// ---- AnalogIO/Outputs/EL4022/EL4022_EX.TcDUT
(*
SPDX-FileCopyrightText: © 2026 Oleksandr Tiutyk <trofimich@gmail.com>
SPDX-License-Identifier: MIT
License: https://opensource.org/license/mit
*)

(*!
<summary>
Beckhoff EL4022_EX: Extended 2-channel analog output terminal (4 .. 20 mA, 12-bit) with diagnostics.
</summary>
<description>
Extends EL4022 with EtherCAT Working Counter, slave state, and CoE mailbox ADS address diagnostics.
When used for I/O, link located fields or their containing buffers to the matching selected PDOs.
The record is not a packed wire buffer; compiler padding is not part of the device specification.
Unlinked/default values do not prove valid I/O. The caller evaluates bus/channel validity before use.
Use one owner task per instance and externally synchronize other access; multi-field snapshots are not atomic.
Copies store data without creating hardware links. Keep borrowed field references valid while consumers are bound.
This passive record performs no validation, synchronization, configuration or protocol advancement.
WcState=TRUE means process-data exchange is invalid. State is acyclic EtherCAT/link information,
not proof of current measurement validity. Link diagnostics to the matching slave InfoData entries.
The selected PDO representation is documented by the base terminal model.
AdsAddr is acyclic mailbox addressing information, not a measurement-validity indicator.
Channels hold raw INT16 output commands; configure electrical range and presentation before use.
</description>
*)
TYPE EL4022_EX EXTENDS EL4022 :
STRUCT
	WcState AT %I* : BOOL;
	State AT %I* : UINT;
	AdsAddr AT %I* : Global.AMSADDR;
END_STRUCT
END_TYPE

// ---- AnalogIO/Outputs/EL4024/EL4024.TcDUT
(*
SPDX-FileCopyrightText: © 2026 Oleksandr Tiutyk <trofimich@gmail.com>
SPDX-License-Identifier: MIT
License: https://opensource.org/license/mit
*)

(*!
<summary>
Beckhoff EL4024: 4-channel analog output terminal (4 .. 20 mA, 12-bit).
</summary>
<description>
Process image mapping structure for the EL4024 EtherCAT terminal with 4 analog output channel(s).
When used for I/O, link located fields or their containing buffers to the matching selected PDOs.
The record is not a packed wire buffer; compiler padding is not part of the device specification.
Unlinked/default values do not prove valid I/O. The caller evaluates bus/channel validity before use.
Use one owner task per instance and externally synchronize other access; multi-field snapshots are not atomic.
Copies store data without creating hardware links. Keep borrowed field references valid while consumers are bound.
This passive record performs no validation, synchronization, configuration or protocol advancement.
Channels hold raw INT16 output commands; configure electrical range and presentation before use.
</description>
*)
TYPE EL4024 :
STRUCT
	Ch1 AT %Q* : INT;
	Ch2 AT %Q* : INT;
	Ch3 AT %Q* : INT;
	Ch4 AT %Q* : INT;
END_STRUCT
END_TYPE

// ---- AnalogIO/Outputs/EL4024/EL4024_EX.TcDUT
(*
SPDX-FileCopyrightText: © 2026 Oleksandr Tiutyk <trofimich@gmail.com>
SPDX-License-Identifier: MIT
License: https://opensource.org/license/mit
*)

(*!
<summary>
Beckhoff EL4024_EX: Extended 4-channel analog output terminal (4 .. 20 mA, 12-bit) with diagnostics.
</summary>
<description>
Extends EL4024 with EtherCAT Working Counter, slave state, and CoE mailbox ADS address diagnostics.
When used for I/O, link located fields or their containing buffers to the matching selected PDOs.
The record is not a packed wire buffer; compiler padding is not part of the device specification.
Unlinked/default values do not prove valid I/O. The caller evaluates bus/channel validity before use.
Use one owner task per instance and externally synchronize other access; multi-field snapshots are not atomic.
Copies store data without creating hardware links. Keep borrowed field references valid while consumers are bound.
This passive record performs no validation, synchronization, configuration or protocol advancement.
WcState=TRUE means process-data exchange is invalid. State is acyclic EtherCAT/link information,
not proof of current measurement validity. Link diagnostics to the matching slave InfoData entries.
The selected PDO representation is documented by the base terminal model.
AdsAddr is acyclic mailbox addressing information, not a measurement-validity indicator.
Channels hold raw INT16 output commands; configure electrical range and presentation before use.
</description>
*)
TYPE EL4024_EX EXTENDS EL4024 :
STRUCT
	WcState AT %I* : BOOL;
	State AT %I* : UINT;
	AdsAddr AT %I* : Global.AMSADDR;
END_STRUCT
END_TYPE

// ---- AnalogIO/Outputs/EL4028/EL4028.TcDUT
(*
SPDX-FileCopyrightText: © 2026 Oleksandr Tiutyk <trofimich@gmail.com>
SPDX-License-Identifier: MIT
License: https://opensource.org/license/mit
*)

(*!
<summary>
Beckhoff EL4028: 8-channel analog output terminal (4 .. 20 mA, 12-bit).
</summary>
<description>
Process image mapping structure for the EL4028 EtherCAT terminal with 8 analog output channel(s).
When used for I/O, link located fields or their containing buffers to the matching selected PDOs.
The record is not a packed wire buffer; compiler padding is not part of the device specification.
Unlinked/default values do not prove valid I/O. The caller evaluates bus/channel validity before use.
Use one owner task per instance and externally synchronize other access; multi-field snapshots are not atomic.
Copies store data without creating hardware links. Keep borrowed field references valid while consumers are bound.
This passive record performs no validation, synchronization, configuration or protocol advancement.
Channels hold raw INT16 output commands; configure electrical range and presentation before use.
</description>
*)
TYPE EL4028 :
STRUCT
	Ch1 AT %Q* : INT;
	Ch2 AT %Q* : INT;
	Ch3 AT %Q* : INT;
	Ch4 AT %Q* : INT;
	Ch5 AT %Q* : INT;
	Ch6 AT %Q* : INT;
	Ch7 AT %Q* : INT;
	Ch8 AT %Q* : INT;
END_STRUCT
END_TYPE

// ---- AnalogIO/Outputs/EL4028/EL4028_EX.TcDUT
(*
SPDX-FileCopyrightText: © 2026 Oleksandr Tiutyk <trofimich@gmail.com>
SPDX-License-Identifier: MIT
License: https://opensource.org/license/mit
*)

(*!
<summary>
Beckhoff EL4028_EX: Extended 8-channel analog output terminal (4 .. 20 mA, 12-bit) with diagnostics.
</summary>
<description>
Extends EL4028 with EtherCAT Working Counter, slave state, and CoE mailbox ADS address diagnostics.
When used for I/O, link located fields or their containing buffers to the matching selected PDOs.
The record is not a packed wire buffer; compiler padding is not part of the device specification.
Unlinked/default values do not prove valid I/O. The caller evaluates bus/channel validity before use.
Use one owner task per instance and externally synchronize other access; multi-field snapshots are not atomic.
Copies store data without creating hardware links. Keep borrowed field references valid while consumers are bound.
This passive record performs no validation, synchronization, configuration or protocol advancement.
WcState=TRUE means process-data exchange is invalid. State is acyclic EtherCAT/link information,
not proof of current measurement validity. Link diagnostics to the matching slave InfoData entries.
The selected PDO representation is documented by the base terminal model.
AdsAddr is acyclic mailbox addressing information, not a measurement-validity indicator.
Channels hold raw INT16 output commands; configure electrical range and presentation before use.
</description>
*)
TYPE EL4028_EX EXTENDS EL4028 :
STRUCT
	WcState AT %I* : BOOL;
	State AT %I* : UINT;
	AdsAddr AT %I* : Global.AMSADDR;
END_STRUCT
END_TYPE

// ---- AnalogIO/Outputs/EL4102/EL4102.TcDUT
(*
SPDX-FileCopyrightText: © 2026 Oleksandr Tiutyk <trofimich@gmail.com>
SPDX-License-Identifier: MIT
License: https://opensource.org/license/mit
*)

(*!
<summary>
Beckhoff EL4102: 2-channel analog output terminal (0 .. 10 V, 16-bit).
</summary>
<description>
Process image mapping structure for the EL4102 EtherCAT terminal with 2 analog output channel(s).
When used for I/O, link located fields or their containing buffers to the matching selected PDOs.
The record is not a packed wire buffer; compiler padding is not part of the device specification.
Unlinked/default values do not prove valid I/O. The caller evaluates bus/channel validity before use.
Use one owner task per instance and externally synchronize other access; multi-field snapshots are not atomic.
Copies store data without creating hardware links. Keep borrowed field references valid while consumers are bound.
This passive record performs no validation, synchronization, configuration or protocol advancement.
Channels hold raw INT16 output commands; configure electrical range and presentation before use.
</description>
*)
TYPE EL4102 :
STRUCT
	Ch1 AT %Q* : INT;
	Ch2 AT %Q* : INT;
END_STRUCT
END_TYPE

// ---- AnalogIO/Outputs/EL4102/EL4102_EX.TcDUT
(*
SPDX-FileCopyrightText: © 2026 Oleksandr Tiutyk <trofimich@gmail.com>
SPDX-License-Identifier: MIT
License: https://opensource.org/license/mit
*)

(*!
<summary>
Beckhoff EL4102_EX: Extended 2-channel analog output terminal (0 .. 10 V, 16-bit) with diagnostics.
</summary>
<description>
Extends EL4102 with EtherCAT Working Counter, slave state, and CoE mailbox ADS address diagnostics.
When used for I/O, link located fields or their containing buffers to the matching selected PDOs.
The record is not a packed wire buffer; compiler padding is not part of the device specification.
Unlinked/default values do not prove valid I/O. The caller evaluates bus/channel validity before use.
Use one owner task per instance and externally synchronize other access; multi-field snapshots are not atomic.
Copies store data without creating hardware links. Keep borrowed field references valid while consumers are bound.
This passive record performs no validation, synchronization, configuration or protocol advancement.
WcState=TRUE means process-data exchange is invalid. State is acyclic EtherCAT/link information,
not proof of current measurement validity. Link diagnostics to the matching slave InfoData entries.
The selected PDO representation is documented by the base terminal model.
AdsAddr is acyclic mailbox addressing information, not a measurement-validity indicator.
Channels hold raw INT16 output commands; configure electrical range and presentation before use.
</description>
*)
TYPE EL4102_EX EXTENDS EL4102 :
STRUCT
	WcState AT %I* : BOOL;
	State AT %I* : UINT;
	AdsAddr AT %I* : Global.AMSADDR;
END_STRUCT
END_TYPE

// ---- AnalogIO/Outputs/EL4104/EL4104.TcDUT
(*
SPDX-FileCopyrightText: © 2026 Oleksandr Tiutyk <trofimich@gmail.com>
SPDX-License-Identifier: MIT
License: https://opensource.org/license/mit
*)

(*!
<summary>
Beckhoff EL4104: 4-channel analog output terminal (0 .. 10 V, 16-bit).
</summary>
<description>
Process image mapping structure for the EL4104 EtherCAT terminal with 4 analog output channel(s).
When used for I/O, link located fields or their containing buffers to the matching selected PDOs.
The record is not a packed wire buffer; compiler padding is not part of the device specification.
Unlinked/default values do not prove valid I/O. The caller evaluates bus/channel validity before use.
Use one owner task per instance and externally synchronize other access; multi-field snapshots are not atomic.
Copies store data without creating hardware links. Keep borrowed field references valid while consumers are bound.
This passive record performs no validation, synchronization, configuration or protocol advancement.
Channels hold raw INT16 output commands; configure electrical range and presentation before use.
</description>
*)
TYPE EL4104 :
STRUCT
	Ch1 AT %Q* : INT;
	Ch2 AT %Q* : INT;
	Ch3 AT %Q* : INT;
	Ch4 AT %Q* : INT;
END_STRUCT
END_TYPE

// ---- AnalogIO/Outputs/EL4104/EL4104_EX.TcDUT
(*
SPDX-FileCopyrightText: © 2026 Oleksandr Tiutyk <trofimich@gmail.com>
SPDX-License-Identifier: MIT
License: https://opensource.org/license/mit
*)

(*!
<summary>
Beckhoff EL4104_EX: Extended 4-channel analog output terminal (0 .. 10 V, 16-bit) with diagnostics.
</summary>
<description>
Extends EL4104 with EtherCAT Working Counter, slave state, and CoE mailbox ADS address diagnostics.
When used for I/O, link located fields or their containing buffers to the matching selected PDOs.
The record is not a packed wire buffer; compiler padding is not part of the device specification.
Unlinked/default values do not prove valid I/O. The caller evaluates bus/channel validity before use.
Use one owner task per instance and externally synchronize other access; multi-field snapshots are not atomic.
Copies store data without creating hardware links. Keep borrowed field references valid while consumers are bound.
This passive record performs no validation, synchronization, configuration or protocol advancement.
WcState=TRUE means process-data exchange is invalid. State is acyclic EtherCAT/link information,
not proof of current measurement validity. Link diagnostics to the matching slave InfoData entries.
The selected PDO representation is documented by the base terminal model.
AdsAddr is acyclic mailbox addressing information, not a measurement-validity indicator.
Channels hold raw INT16 output commands; configure electrical range and presentation before use.
</description>
*)
TYPE EL4104_EX EXTENDS EL4104 :
STRUCT
	WcState AT %I* : BOOL;
	State AT %I* : UINT;
	AdsAddr AT %I* : Global.AMSADDR;
END_STRUCT
END_TYPE

// ---- AnalogIO/Outputs/EL4132/EL4132.TcDUT
(*
SPDX-FileCopyrightText: © 2026 Oleksandr Tiutyk <trofimich@gmail.com>
SPDX-License-Identifier: MIT
License: https://opensource.org/license/mit
*)

(*!
<summary>
Beckhoff EL4132: 2-channel analog output terminal (-10 V .. +10 V, 16-bit).
</summary>
<description>
Process image mapping structure for the EL4132 EtherCAT terminal with 2 analog output channel(s).
When used for I/O, link located fields or their containing buffers to the matching selected PDOs.
The record is not a packed wire buffer; compiler padding is not part of the device specification.
Unlinked/default values do not prove valid I/O. The caller evaluates bus/channel validity before use.
Use one owner task per instance and externally synchronize other access; multi-field snapshots are not atomic.
Copies store data without creating hardware links. Keep borrowed field references valid while consumers are bound.
This passive record performs no validation, synchronization, configuration or protocol advancement.
Channels hold raw INT16 output commands; configure electrical range and presentation before use.
</description>
*)
TYPE EL4132 :
STRUCT
	Ch1 AT %Q* : INT;
	Ch2 AT %Q* : INT;
END_STRUCT
END_TYPE

// ---- AnalogIO/Outputs/EL4132/EL4132_EX.TcDUT
(*
SPDX-FileCopyrightText: © 2026 Oleksandr Tiutyk <trofimich@gmail.com>
SPDX-License-Identifier: MIT
License: https://opensource.org/license/mit
*)

(*!
<summary>
Beckhoff EL4132_EX: Extended 2-channel analog output terminal (-10 V .. +10 V, 16-bit) with diagnostics.
</summary>
<description>
Extends EL4132 with EtherCAT Working Counter, slave state, and CoE mailbox ADS address diagnostics.
When used for I/O, link located fields or their containing buffers to the matching selected PDOs.
The record is not a packed wire buffer; compiler padding is not part of the device specification.
Unlinked/default values do not prove valid I/O. The caller evaluates bus/channel validity before use.
Use one owner task per instance and externally synchronize other access; multi-field snapshots are not atomic.
Copies store data without creating hardware links. Keep borrowed field references valid while consumers are bound.
This passive record performs no validation, synchronization, configuration or protocol advancement.
WcState=TRUE means process-data exchange is invalid. State is acyclic EtherCAT/link information,
not proof of current measurement validity. Link diagnostics to the matching slave InfoData entries.
The selected PDO representation is documented by the base terminal model.
AdsAddr is acyclic mailbox addressing information, not a measurement-validity indicator.
Channels hold raw INT16 output commands; configure electrical range and presentation before use.
</description>
*)
TYPE EL4132_EX EXTENDS EL4132 :
STRUCT
	WcState AT %I* : BOOL;
	State AT %I* : UINT;
	AdsAddr AT %I* : Global.AMSADDR;
END_STRUCT
END_TYPE

// ---- AnalogIO/Outputs/EL4134/EL4134.TcDUT
(*
SPDX-FileCopyrightText: © 2026 Oleksandr Tiutyk <trofimich@gmail.com>
SPDX-License-Identifier: MIT
License: https://opensource.org/license/mit
*)

(*!
<summary>
Beckhoff EL4134: 4-channel analog output terminal (-10 V .. +10 V, 16-bit).
</summary>
<description>
Process image mapping structure for the EL4134 EtherCAT terminal with 4 analog output channel(s).
When used for I/O, link located fields or their containing buffers to the matching selected PDOs.
The record is not a packed wire buffer; compiler padding is not part of the device specification.
Unlinked/default values do not prove valid I/O. The caller evaluates bus/channel validity before use.
Use one owner task per instance and externally synchronize other access; multi-field snapshots are not atomic.
Copies store data without creating hardware links. Keep borrowed field references valid while consumers are bound.
This passive record performs no validation, synchronization, configuration or protocol advancement.
Channels hold raw INT16 output commands; configure electrical range and presentation before use.
</description>
*)
TYPE EL4134 :
STRUCT
	Ch1 AT %Q* : INT;
	Ch2 AT %Q* : INT;
	Ch3 AT %Q* : INT;
	Ch4 AT %Q* : INT;
END_STRUCT
END_TYPE

// ---- AnalogIO/Outputs/EL4134/EL4134_EX.TcDUT
(*
SPDX-FileCopyrightText: © 2026 Oleksandr Tiutyk <trofimich@gmail.com>
SPDX-License-Identifier: MIT
License: https://opensource.org/license/mit
*)

(*!
<summary>
Beckhoff EL4134_EX: Extended 4-channel analog output terminal (-10 V .. +10 V, 16-bit) with diagnostics.
</summary>
<description>
Extends EL4134 with EtherCAT Working Counter, slave state, and CoE mailbox ADS address diagnostics.
When used for I/O, link located fields or their containing buffers to the matching selected PDOs.
The record is not a packed wire buffer; compiler padding is not part of the device specification.
Unlinked/default values do not prove valid I/O. The caller evaluates bus/channel validity before use.
Use one owner task per instance and externally synchronize other access; multi-field snapshots are not atomic.
Copies store data without creating hardware links. Keep borrowed field references valid while consumers are bound.
This passive record performs no validation, synchronization, configuration or protocol advancement.
WcState=TRUE means process-data exchange is invalid. State is acyclic EtherCAT/link information,
not proof of current measurement validity. Link diagnostics to the matching slave InfoData entries.
The selected PDO representation is documented by the base terminal model.
AdsAddr is acyclic mailbox addressing information, not a measurement-validity indicator.
Channels hold raw INT16 output commands; configure electrical range and presentation before use.
</description>
*)
TYPE EL4134_EX EXTENDS EL4134 :
STRUCT
	WcState AT %I* : BOOL;
	State AT %I* : UINT;
	AdsAddr AT %I* : Global.AMSADDR;
END_STRUCT
END_TYPE

// ---- AnalogIO/Outputs/EL4122/EL4122.TcDUT
(*
SPDX-FileCopyrightText: © 2026 Oleksandr Tiutyk <trofimich@gmail.com>
SPDX-License-Identifier: MIT
License: https://opensource.org/license/mit
*)

(*!
<summary>
Beckhoff EL4122: 2-channel analog output terminal (4 .. 20 mA, 16-bit).
</summary>
<description>
Process image mapping structure for the EL4122 EtherCAT terminal with 2 analog output channel(s).
When used for I/O, link located fields or their containing buffers to the matching selected PDOs.
The record is not a packed wire buffer; compiler padding is not part of the device specification.
Unlinked/default values do not prove valid I/O. The caller evaluates bus/channel validity before use.
Use one owner task per instance and externally synchronize other access; multi-field snapshots are not atomic.
Copies store data without creating hardware links. Keep borrowed field references valid while consumers are bound.
This passive record performs no validation, synchronization, configuration or protocol advancement.
Channels hold raw INT16 output commands; configure electrical range and presentation before use.
</description>
*)
TYPE EL4122 :
STRUCT
	Ch1 AT %Q* : INT;
	Ch2 AT %Q* : INT;
END_STRUCT
END_TYPE

// ---- AnalogIO/Outputs/EL4122/EL4122_EX.TcDUT
(*
SPDX-FileCopyrightText: © 2026 Oleksandr Tiutyk <trofimich@gmail.com>
SPDX-License-Identifier: MIT
License: https://opensource.org/license/mit
*)

(*!
<summary>
Beckhoff EL4122_EX: Extended 2-channel analog output terminal (4 .. 20 mA, 16-bit) with diagnostics.
</summary>
<description>
Extends EL4122 with EtherCAT Working Counter, slave state, and CoE mailbox ADS address diagnostics.
When used for I/O, link located fields or their containing buffers to the matching selected PDOs.
The record is not a packed wire buffer; compiler padding is not part of the device specification.
Unlinked/default values do not prove valid I/O. The caller evaluates bus/channel validity before use.
Use one owner task per instance and externally synchronize other access; multi-field snapshots are not atomic.
Copies store data without creating hardware links. Keep borrowed field references valid while consumers are bound.
This passive record performs no validation, synchronization, configuration or protocol advancement.
WcState=TRUE means process-data exchange is invalid. State is acyclic EtherCAT/link information,
not proof of current measurement validity. Link diagnostics to the matching slave InfoData entries.
The selected PDO representation is documented by the base terminal model.
AdsAddr is acyclic mailbox addressing information, not a measurement-validity indicator.
Channels hold raw INT16 output commands; configure electrical range and presentation before use.
</description>
*)
TYPE EL4122_EX EXTENDS EL4122 :
STRUCT
	WcState AT %I* : BOOL;
	State AT %I* : UINT;
	AdsAddr AT %I* : Global.AMSADDR;
END_STRUCT
END_TYPE

// ---- AnalogIO/Outputs/EL4124/EL4124.TcDUT
(*
SPDX-FileCopyrightText: © 2026 Oleksandr Tiutyk <trofimich@gmail.com>
SPDX-License-Identifier: MIT
License: https://opensource.org/license/mit
*)

(*!
<summary>
Beckhoff EL4124: 4-channel analog output terminal (4 .. 20 mA, 16-bit).
</summary>
<description>
Process image mapping structure for the EL4124 EtherCAT terminal with 4 analog output channel(s).
When used for I/O, link located fields or their containing buffers to the matching selected PDOs.
The record is not a packed wire buffer; compiler padding is not part of the device specification.
Unlinked/default values do not prove valid I/O. The caller evaluates bus/channel validity before use.
Use one owner task per instance and externally synchronize other access; multi-field snapshots are not atomic.
Copies store data without creating hardware links. Keep borrowed field references valid while consumers are bound.
This passive record performs no validation, synchronization, configuration or protocol advancement.
Channels hold raw INT16 output commands; configure electrical range and presentation before use.
</description>
*)
TYPE EL4124 :
STRUCT
	Ch1 AT %Q* : INT;
	Ch2 AT %Q* : INT;
	Ch3 AT %Q* : INT;
	Ch4 AT %Q* : INT;
END_STRUCT
END_TYPE

// ---- AnalogIO/Outputs/EL4124/EL4124_EX.TcDUT
(*
SPDX-FileCopyrightText: © 2026 Oleksandr Tiutyk <trofimich@gmail.com>
SPDX-License-Identifier: MIT
License: https://opensource.org/license/mit
*)

(*!
<summary>
Beckhoff EL4124_EX: Extended 4-channel analog output terminal (4 .. 20 mA, 16-bit) with diagnostics.
</summary>
<description>
Extends EL4124 with EtherCAT Working Counter, slave state, and CoE mailbox ADS address diagnostics.
When used for I/O, link located fields or their containing buffers to the matching selected PDOs.
The record is not a packed wire buffer; compiler padding is not part of the device specification.
Unlinked/default values do not prove valid I/O. The caller evaluates bus/channel validity before use.
Use one owner task per instance and externally synchronize other access; multi-field snapshots are not atomic.
Copies store data without creating hardware links. Keep borrowed field references valid while consumers are bound.
This passive record performs no validation, synchronization, configuration or protocol advancement.
WcState=TRUE means process-data exchange is invalid. State is acyclic EtherCAT/link information,
not proof of current measurement validity. Link diagnostics to the matching slave InfoData entries.
The selected PDO representation is documented by the base terminal model.
AdsAddr is acyclic mailbox addressing information, not a measurement-validity indicator.
Channels hold raw INT16 output commands; configure electrical range and presentation before use.
</description>
*)
TYPE EL4124_EX EXTENDS EL4124 :
STRUCT
	WcState AT %I* : BOOL;
	State AT %I* : UINT;
	AdsAddr AT %I* : Global.AMSADDR;
END_STRUCT
END_TYPE

// ---- Weighing/STRAIN_GAUGE_INPUT_CHANNEL.TcDUT
(*
SPDX-FileCopyrightText: © 2026 Oleksandr Tiutyk <trofimich@gmail.com>
SPDX-License-Identifier: MIT
License: https://opensource.org/license/mit
*)

(*!
<summary>
Beckhoff strain gauge / resistor bridge input channel process image.
</summary>
<description>
Represents EL3356/EL3356-0010 input PDO 0x1A00 with 16-bit Status and PDO 0x1A01 with signed 32-bit Value.
Both input PDOs are required. Link Status to RMB Status and Value to RMB Value (INT32) separately;
PDO 0x1A01 alone does not contain status information.
Select the integer assignment; REAL load and two-channel voltage modes require different types.
Calibration and device settings determine engineering scaling. Evaluate Status before using Value.
When used for I/O, link located fields or their containing buffers to the matching selected PDOs.
The record is not a packed wire buffer; compiler padding is not part of the device specification.
Unlinked/default values do not prove valid I/O. The caller evaluates bus/channel validity before use.
Use one owner task per instance and externally synchronize other access; multi-field snapshots are not atomic.
Copies store data without creating hardware links. Keep borrowed field references valid while consumers are bound.
This passive record performs no validation, synchronization, configuration or protocol advancement.
</description>
*)
TYPE STRAIN_GAUGE_INPUT_CHANNEL :
STRUCT
	Status AT %I* : WORD;
	Value AT %I* : DINT;
END_STRUCT
END_TYPE

// ---- Weighing/STRAIN_GAUGE_OUTPUT_CHANNEL.TcDUT
(*
SPDX-FileCopyrightText: © 2026 Oleksandr Tiutyk <trofimich@gmail.com>
SPDX-License-Identifier: MIT
License: https://opensource.org/license/mit
*)

(*!
<summary>
Beckhoff strain gauge / resistor bridge output control channel process image.
</summary>
<description>
Encapsulates a 16-bit control word for calibration, tare, and filtering commands on measuring bridge terminals
(e.g. EL3356).
When used for I/O, link located fields or their containing buffers to the matching selected PDOs.
The record is not a packed wire buffer; compiler padding is not part of the device specification.
Unlinked/default values do not prove valid I/O. The caller evaluates bus/channel validity before use.
Use one owner task per instance and externally synchronize other access; multi-field snapshots are not atomic.
Copies store data without creating hardware links. Keep borrowed field references valid while consumers are bound.
This passive record performs no validation, synchronization, configuration or protocol advancement.
</description>
*)
TYPE STRAIN_GAUGE_OUTPUT_CHANNEL :
STRUCT
	Control AT %Q* : WORD;
END_STRUCT
END_TYPE

// ---- Weighing/STRAIN_GAUGE_CHANNEL.TcDUT
(*
SPDX-FileCopyrightText: © 2026 Oleksandr Tiutyk <trofimich@gmail.com>
SPDX-License-Identifier: MIT
License: https://opensource.org/license/mit
*)

(*!
<summary>
Beckhoff bidirectional strain gauge / resistor bridge channel process image.
</summary>
<description>
Aggregates input status/value (STRAIN_GAUGE_INPUT_CHANNEL) and output control (STRAIN_GAUGE_OUTPUT_CHANNEL)
for one measuring bridge channel.
When used for I/O, link located fields or their containing buffers to the matching selected PDOs.
The record is not a packed wire buffer; compiler padding is not part of the device specification.
Unlinked/default values do not prove valid I/O. The caller evaluates bus/channel validity before use.
Use one owner task per instance and externally synchronize other access; multi-field snapshots are not atomic.
Copies store data without creating hardware links. Keep borrowed field references valid while consumers are bound.
This passive record performs no validation, synchronization, configuration or protocol advancement.
</description>
*)
TYPE STRAIN_GAUGE_CHANNEL :
STRUCT
	In : STRAIN_GAUGE_INPUT_CHANNEL;
	Out : STRAIN_GAUGE_OUTPUT_CHANNEL;
END_STRUCT
END_TYPE

// ---- Weighing/EL3356/EL3356.TcDUT
(*
SPDX-FileCopyrightText: © 2026 Oleksandr Tiutyk <trofimich@gmail.com>
SPDX-License-Identifier: MIT
License: https://opensource.org/license/mit
*)

(*!
<summary>
Beckhoff EL3356: 1-channel precise resistor bridge / load cell terminal (24-bit).
</summary>
<description>
Requires the one-channel strain-gauge INT32 assignment: status PDO 0x1A00, value PDO 0x1A01,
and control PDO 0x1600. Keep both input PDOs enabled and link Status and Value separately.
Value is signed calculated load; engineering scaling follows calibration. REAL load, two-channel voltage,
optional filter-frequency and timestamp PDOs are outside this model; disable or link optional PDOs separately.
When used for I/O, link located fields or their containing buffers to the matching selected PDOs.
The record is not a packed wire buffer; compiler padding is not part of the device specification.
Unlinked/default values do not prove valid I/O. The caller evaluates bus/channel validity before use.
Use one owner task per instance and externally synchronize other access; multi-field snapshots are not atomic.
Copies store data without creating hardware links. Keep borrowed field references valid while consumers are bound.
This passive record performs no validation, synchronization, configuration or protocol advancement.
</description>
*)
TYPE EL3356 :
STRUCT
	Ch1 : STRAIN_GAUGE_CHANNEL;
END_STRUCT
END_TYPE

// ---- Weighing/EL3356/EL3356_EX.TcDUT
(*
SPDX-FileCopyrightText: © 2026 Oleksandr Tiutyk <trofimich@gmail.com>
SPDX-License-Identifier: MIT
License: https://opensource.org/license/mit
*)

(*!
<summary>
Beckhoff EL3356_EX: Extended 1-channel load cell terminal with diagnostics.
</summary>
<description>
Extends EL3356 with EtherCAT Working Counter, slave state, and CoE mailbox ADS address diagnostics.
When used for I/O, link located fields or their containing buffers to the matching selected PDOs.
The record is not a packed wire buffer; compiler padding is not part of the device specification.
Unlinked/default values do not prove valid I/O. The caller evaluates bus/channel validity before use.
Use one owner task per instance and externally synchronize other access; multi-field snapshots are not atomic.
Copies store data without creating hardware links. Keep borrowed field references valid while consumers are bound.
This passive record performs no validation, synchronization, configuration or protocol advancement.
WcState=TRUE means process-data exchange is invalid. State is acyclic EtherCAT/link information,
not proof of current measurement validity. Link diagnostics to the matching slave InfoData entries.
The selected PDO representation is documented by the base terminal model.
InputToggle signals an input update by changing state; TRUE alone does not mean fresh data.
AdsAddr is acyclic mailbox addressing information, not a measurement-validity indicator.
</description>
*)
TYPE EL3356_EX EXTENDS EL3356 :
STRUCT
	WcState AT %I* : BOOL;
	InputToggle AT %I* : BOOL;
	State AT %I* : UINT;
	AdsAddr AT %I* : Global.AMSADDR;
END_STRUCT
END_TYPE

// ---- Weighing/EL3356_0010/EL3356_0010.TcDUT
(*
SPDX-FileCopyrightText: © 2026 Oleksandr Tiutyk <trofimich@gmail.com>
SPDX-License-Identifier: MIT
License: https://opensource.org/license/mit
*)

(*!
<summary>
Beckhoff EL3356-0010: Fast 1-channel precise resistor bridge / load cell terminal with Distributed Clocks.
</summary>
<description>
Requires the one-channel strain-gauge INT32 assignment: status PDO 0x1A00, value PDO 0x1A01,
and control PDO 0x1600. Keep both input PDOs enabled and link Status and Value separately.
Value is signed calculated load; engineering scaling follows calibration. REAL load, two-channel voltage,
optional filter-frequency and timestamp PDOs are outside this model; disable or link optional PDOs separately.
When used for I/O, link located fields or their containing buffers to the matching selected PDOs.
The record is not a packed wire buffer; compiler padding is not part of the device specification.
Unlinked/default values do not prove valid I/O. The caller evaluates bus/channel validity before use.
Use one owner task per instance and externally synchronize other access; multi-field snapshots are not atomic.
Copies store data without creating hardware links. Keep borrowed field references valid while consumers are bound.
This passive record performs no validation, synchronization, configuration or protocol advancement.
</description>
*)
TYPE EL3356_0010 :
STRUCT
	Ch1 : STRAIN_GAUGE_CHANNEL;
END_STRUCT
END_TYPE

// ---- Weighing/EL3356_0010/EL3356_0010_EX.TcDUT
(*
SPDX-FileCopyrightText: © 2026 Oleksandr Tiutyk <trofimich@gmail.com>
SPDX-License-Identifier: MIT
License: https://opensource.org/license/mit
*)

(*!
<summary>
Beckhoff EL3356_0010_EX: Extended fast 1-channel load cell terminal with diagnostics.
</summary>
<description>
Extends EL3356_0010 with EtherCAT Working Counter, slave state, and CoE mailbox ADS address diagnostics.
When used for I/O, link located fields or their containing buffers to the matching selected PDOs.
The record is not a packed wire buffer; compiler padding is not part of the device specification.
Unlinked/default values do not prove valid I/O. The caller evaluates bus/channel validity before use.
Use one owner task per instance and externally synchronize other access; multi-field snapshots are not atomic.
Copies store data without creating hardware links. Keep borrowed field references valid while consumers are bound.
This passive record performs no validation, synchronization, configuration or protocol advancement.
WcState=TRUE means process-data exchange is invalid. State is acyclic EtherCAT/link information,
not proof of current measurement validity. Link diagnostics to the matching slave InfoData entries.
The selected PDO representation is documented by the base terminal model.
InputToggle signals an input update by changing state; TRUE alone does not mean fresh data.
AdsAddr is acyclic mailbox addressing information, not a measurement-validity indicator.
</description>
*)
TYPE EL3356_0010_EX EXTENDS EL3356_0010 :
STRUCT
	WcState AT %I* : BOOL;
	InputToggle AT %I* : BOOL;
	State AT %I* : UINT;
	AdsAddr AT %I* : Global.AMSADDR;
END_STRUCT
END_TYPE

// ---- PowerMeasurement/POWER_MEASUREMENT_INPUT_CHANNEL.TcDUT
(*
SPDX-FileCopyrightText: © 2026 Oleksandr Tiutyk <trofimich@gmail.com>
SPDX-License-Identifier: MIT
License: https://opensource.org/license/mit
*)

(*!
<summary>
Beckhoff 3-phase power measurement input channel process image.
</summary>
<description>
Represents EL3413/EL3433 phase PDO 0x1A00, 0x1A01 or 0x1A02, including mandatory channel Status.
Status contains voltage/current limits, phase sequence, missing zero crossing, TxPDO State and Toggle.
Reject data when Status bit 14 is set; bit 15 toggles on update. Evaluate bus validity as well.
Current is signed in 0.000001 A, Voltage in 0.0001 V and ActivePower in 0.01 W before transformer ratios.
Index acknowledges the selection for VariantValue; do not interpret it using only the requested output Index.
Indices 0..5 select apparent power (0.01 VA), reactive power (0.01 var), energy (0.001 Wh), power factor
(0.001), frequency (0.1 Hz) and negative energy (0.001 Wh). Further indices depend on device firmware.
EL3403 uses EL3403_INPUT_CHANNEL because its phase status differs. Link fields individually, not as a wire buffer.
Use one owner task and synchronize other access; copies do not guarantee an atomic snapshot.
When used for I/O, link located fields or their containing buffers to the matching selected PDOs.
The record is not a packed wire buffer; compiler padding is not part of the device specification.
Unlinked/default values do not prove valid I/O. The caller evaluates bus/channel validity before use.
Use one owner task per instance and externally synchronize other access; multi-field snapshots are not atomic.
Copies store data without creating hardware links. Keep borrowed field references valid while consumers are bound.
This passive record performs no validation, synchronization, configuration or protocol advancement.
</description>
*)
TYPE POWER_MEASUREMENT_INPUT_CHANNEL :
STRUCT
	//! <summary>Phase status; TxPDO State bit 14 invalidates data and bit 15 toggles on update.</summary>
	Status AT %I* : WORD;
	Current AT %I* : DINT;
	Voltage AT %I* : DINT;
	ActivePower AT %I* : DINT;
	Index AT %I* : USINT;
	VariantValue AT %I* : DINT;
END_STRUCT
END_TYPE

// ---- PowerMeasurement/POWER_MEASUREMENT_OUTPUT_CHANNEL.TcDUT
(*
SPDX-FileCopyrightText: © 2026 Oleksandr Tiutyk <trofimich@gmail.com>
SPDX-License-Identifier: MIT
License: https://opensource.org/license/mit
*)

(*!
<summary>
Beckhoff 3-phase power measurement output control channel process image.
</summary>
<description>
One UINT8 Index selector at 0x7000:01, 0x7010:01 or 0x7020:01.
Common indices 0..5 select apparent power, reactive power, energy, power factor, frequency and negative energy.
Other indices depend on terminal/firmware. Wait for input acknowledgement and valid status before interpreting
VariantValue; a selector write is not a synchronous measurement read. Use one owner task for output writes.
When used for I/O, link located fields or their containing buffers to the matching selected PDOs.
The record is not a packed wire buffer; compiler padding is not part of the device specification.
Unlinked/default values do not prove valid I/O. The caller evaluates bus/channel validity before use.
Use one owner task per instance and externally synchronize other access; multi-field snapshots are not atomic.
Copies store data without creating hardware links. Keep borrowed field references valid while consumers are bound.
This passive record performs no validation, synchronization, configuration or protocol advancement.
</description>
*)
TYPE POWER_MEASUREMENT_OUTPUT_CHANNEL :
STRUCT
	Index AT %Q* : USINT;
END_STRUCT
END_TYPE

// ---- PowerMeasurement/POWER_MEASUREMENT_CHANNEL.TcDUT
(*
SPDX-FileCopyrightText: © 2026 Oleksandr Tiutyk <trofimich@gmail.com>
SPDX-License-Identifier: MIT
License: https://opensource.org/license/mit
*)

(*!
<summary>
Beckhoff bidirectional power measurement phase channel process image.
</summary>
<description>
Combines an EL3413/EL3433 phase input PDO, including mandatory Status, with its output Index selector.
Evaluate input validity and wait for In.Index to acknowledge Out.Index before interpreting In.VariantValue.
EL3403 uses EL3403_CHANNEL; its phase status flags are different. Link input/output fields individually.
Use one owner task and synchronize other access; copying stores data without creating new hardware links.
When used for I/O, link located fields or their containing buffers to the matching selected PDOs.
The record is not a packed wire buffer; compiler padding is not part of the device specification.
Unlinked/default values do not prove valid I/O. The caller evaluates bus/channel validity before use.
Use one owner task per instance and externally synchronize other access; multi-field snapshots are not atomic.
Copies store data without creating hardware links. Keep borrowed field references valid while consumers are bound.
This passive record performs no validation, synchronization, configuration or protocol advancement.
</description>
*)
TYPE POWER_MEASUREMENT_CHANNEL :
STRUCT
	In : POWER_MEASUREMENT_INPUT_CHANNEL;
	Out : POWER_MEASUREMENT_OUTPUT_CHANNEL;
END_STRUCT
END_TYPE

// ---- PowerMeasurement/POWER_MEASUREMENT_AUXILIARY_INPUT_CHANNEL.TcDUT
(*
SPDX-FileCopyrightText: © 2026 Oleksandr Tiutyk <trofimich@gmail.com>
SPDX-License-Identifier: MIT
License: https://opensource.org/license/mit
*)

(*!
<summary>Beckhoff EL3413/EL3433 auxiliary measurement input PDO.</summary>
<description>
Represents TxPDO 0x1A03 at 0x6030: Status WORD, acknowledged Index/Channel bytes and signed Value.
Status bit 2 reports overcurrent where supported, bit 14 invalidates data and bit 15 toggles on update.
Use Value only after both input selectors acknowledge the requested output selectors and status is valid.
Units and supported selector combinations depend on device/firmware; examples include neutral current,
energy totals and harmonics. This raw record performs no unit conversion or validity checking.
Link fields individually. Use one owner task and synchronize other access; snapshots are not atomic.
When used for I/O, link located fields or their containing buffers to the matching selected PDOs.
The record is not a packed wire buffer; compiler padding is not part of the device specification.
Unlinked/default values do not prove valid I/O. The caller evaluates bus/channel validity before use.
Use one owner task per instance and externally synchronize other access; multi-field snapshots are not atomic.
Copies store data without creating hardware links. Keep borrowed field references valid while consumers are bound.
This passive record performs no validation, synchronization, configuration or protocol advancement.
</description>
*)
TYPE POWER_MEASUREMENT_AUXILIARY_INPUT_CHANNEL :
STRUCT
	Status AT %I* : WORD;
	Index AT %I* : USINT;
	Channel AT %I* : USINT;
	Value AT %I* : DINT;
END_STRUCT
END_TYPE

// ---- PowerMeasurement/POWER_MEASUREMENT_AUXILIARY_OUTPUT_CHANNEL.TcDUT
(*
SPDX-FileCopyrightText: © 2026 Oleksandr Tiutyk <trofimich@gmail.com>
SPDX-License-Identifier: MIT
License: https://opensource.org/license/mit
*)

(*!
<summary>Beckhoff EL3413/EL3433 auxiliary measurement selectors.</summary>
<description>
Represents RxPDO 0x1603: Index at 0x7030:01 and Channel at 0x7030:02, both UINT8.
Select a combination supported by the device/firmware. Selection takes effect asynchronously;
wait for both acknowledged input selectors and valid input status before interpreting auxiliary Value.
Link fields individually and use one owner task for writes; externally synchronize other access.
When used for I/O, link located fields or their containing buffers to the matching selected PDOs.
The record is not a packed wire buffer; compiler padding is not part of the device specification.
Unlinked/default values do not prove valid I/O. The caller evaluates bus/channel validity before use.
Use one owner task per instance and externally synchronize other access; multi-field snapshots are not atomic.
Copies store data without creating hardware links. Keep borrowed field references valid while consumers are bound.
This passive record performs no validation, synchronization, configuration or protocol advancement.
</description>
*)
TYPE POWER_MEASUREMENT_AUXILIARY_OUTPUT_CHANNEL :
STRUCT
	Index AT %Q* : USINT;
	Channel AT %Q* : USINT;
END_STRUCT
END_TYPE

// ---- PowerMeasurement/POWER_MEASUREMENT_AUXILIARY_CHANNEL.TcDUT
(*
SPDX-FileCopyrightText: © 2026 Oleksandr Tiutyk <trofimich@gmail.com>
SPDX-License-Identifier: MIT
License: https://opensource.org/license/mit
*)

(*!
<summary>Beckhoff EL3413/EL3433 bidirectional auxiliary measurement channel.</summary>
<description>
Combines auxiliary TxPDO 0x1A03 and selector RxPDO 0x1603 in the represented default process image.
Input status and selector acknowledgements determine when Value can be interpreted for the requested quantity.
This interface is not present in EL3403. Link fields individually; this is not a packed EtherCAT packet.
Use one owner task; externally synchronize other access. Copies store data without creating hardware links.
When used for I/O, link located fields or their containing buffers to the matching selected PDOs.
The record is not a packed wire buffer; compiler padding is not part of the device specification.
Unlinked/default values do not prove valid I/O. The caller evaluates bus/channel validity before use.
Use one owner task per instance and externally synchronize other access; multi-field snapshots are not atomic.
Copies store data without creating hardware links. Keep borrowed field references valid while consumers are bound.
This passive record performs no validation, synchronization, configuration or protocol advancement.
</description>
*)
TYPE POWER_MEASUREMENT_AUXILIARY_CHANNEL :
STRUCT
	In : POWER_MEASUREMENT_AUXILIARY_INPUT_CHANNEL;
	Out : POWER_MEASUREMENT_AUXILIARY_OUTPUT_CHANNEL;
END_STRUCT
END_TYPE

// ---- PowerMeasurement/EL3403/EL3403.TcDUT
(*
SPDX-FileCopyrightText: © 2026 Oleksandr Tiutyk <trofimich@gmail.com>
SPDX-License-Identifier: MIT
License: https://opensource.org/license/mit
*)

(*!
<summary>
Beckhoff EL3403: 3-phase power measurement terminal up to 500 V AC (1 A / 5 A external CT).
</summary>
<description>
Represents phase TxPDOs 0x1A00..0x1A02, terminal Status TxPDO 0x1A03 and selector RxPDOs 0x1600..0x1602.
All status endpoints are required. Phase headers carry sync error/toggle; terminal Status carries missing
zero crossings, phase sequence error and sync error. Evaluate these alongside bus WcState.
Use each input Index acknowledgement to interpret VariantValue; State=OP alone does not validate a measurement.
Link fields individually. Use one owner task and externally synchronize other access; snapshots are not atomic.
When used for I/O, link located fields or their containing buffers to the matching selected PDOs.
The record is not a packed wire buffer; compiler padding is not part of the device specification.
Unlinked/default values do not prove valid I/O. The caller evaluates bus/channel validity before use.
Use one owner task per instance and externally synchronize other access; multi-field snapshots are not atomic.
Copies store data without creating hardware links. Keep borrowed field references valid while consumers are bound.
This passive record performs no validation, synchronization, configuration or protocol advancement.
</description>
*)
TYPE EL3403 :
STRUCT
	L1 : EL3403_CHANNEL;
	L2 : EL3403_CHANNEL;
	L3 : EL3403_CHANNEL;
	//! <summary>TxPDO 0x1A03: missing zero crossings bits 3..5, phase error bit 8 and sync error bit 13.</summary>
	Status AT %I* : WORD;
END_STRUCT
END_TYPE

// ---- PowerMeasurement/EL3403/EL3403_INPUT_CHANNEL.TcDUT
(*
SPDX-FileCopyrightText: © 2026 Oleksandr Tiutyk <trofimich@gmail.com>
SPDX-License-Identifier: MIT
License: https://opensource.org/license/mit
*)

(*!
<summary>Beckhoff EL3403 phase input PDO with synchronization diagnostics.</summary>
<description>
Represents one EL3403 phase TxPDO (0x1A00, 0x1A01 or 0x1A02).
Status is the 16-bit PDO header: bit 13 is Sync error and bit 15 is TxPDO Toggle.
This header does not expose the EL3413/EL3433 voltage/current error flags.
Current and Voltage are signed raw values in 0.000001 A and 0.0001 V; ActivePower is in 0.01 W.
Transformer ratios and terminal variants affect scaling. VariantValue units follow acknowledged Index.
Indices 0..5 select apparent/reactive power, energy, power factor, frequency and negative energy.
Evaluate bus validity, synchronization and terminal-wide Status before using measurements.
Link fields individually; this is not a packed wire buffer. Use one owner task and synchronize other access.
When used for I/O, link located fields or their containing buffers to the matching selected PDOs.
The record is not a packed wire buffer; compiler padding is not part of the device specification.
Unlinked/default values do not prove valid I/O. The caller evaluates bus/channel validity before use.
Use one owner task per instance and externally synchronize other access; multi-field snapshots are not atomic.
Copies store data without creating hardware links. Keep borrowed field references valid while consumers are bound.
This passive record performs no validation, synchronization, configuration or protocol advancement.
</description>
*)
TYPE EL3403_INPUT_CHANNEL :
STRUCT
	Status AT %I* : WORD;
	Current AT %I* : DINT;
	Voltage AT %I* : DINT;
	ActivePower AT %I* : DINT;
	Index AT %I* : USINT;
	VariantValue AT %I* : DINT;
END_STRUCT
END_TYPE

// ---- PowerMeasurement/EL3403/EL3403_CHANNEL.TcDUT
(*
SPDX-FileCopyrightText: © 2026 Oleksandr Tiutyk <trofimich@gmail.com>
SPDX-License-Identifier: MIT
License: https://opensource.org/license/mit
*)

(*!
<summary>Beckhoff EL3403 phase channel with its own input status semantics.</summary>
<description>
Combines EL3403 phase feedback and the output variable-value selector.
Input Index acknowledges output Index; evaluate phase and terminal-wide diagnostics before using values.
Do not substitute POWER_MEASUREMENT_CHANNEL: its input status belongs to EL3413/EL3433.
Link input/output fields individually. Use one owner task and synchronize other access.
Copies store data only; they create no hardware links and do not guarantee an atomic snapshot.
When used for I/O, link located fields or their containing buffers to the matching selected PDOs.
The record is not a packed wire buffer; compiler padding is not part of the device specification.
Unlinked/default values do not prove valid I/O. The caller evaluates bus/channel validity before use.
Use one owner task per instance and externally synchronize other access; multi-field snapshots are not atomic.
Copies store data without creating hardware links. Keep borrowed field references valid while consumers are bound.
This passive record performs no validation, synchronization, configuration or protocol advancement.
</description>
*)
TYPE EL3403_CHANNEL :
STRUCT
	In : EL3403_INPUT_CHANNEL;
	Out : POWER_MEASUREMENT_OUTPUT_CHANNEL;
END_STRUCT
END_TYPE

// ---- PowerMeasurement/EL3403/EL3403_EX.TcDUT
(*
SPDX-FileCopyrightText: © 2026 Oleksandr Tiutyk <trofimich@gmail.com>
SPDX-License-Identifier: MIT
License: https://opensource.org/license/mit
*)

(*!
<summary>
Beckhoff EL3403_EX: Extended 3-phase power measurement terminal up to 500 V AC (1 A / 5 A external CT) with
diagnostics.
</summary>
<description>
Extends EL3403 with EtherCAT Working Counter, slave state, and CoE mailbox ADS address diagnostics.
When used for I/O, link located fields or their containing buffers to the matching selected PDOs.
The record is not a packed wire buffer; compiler padding is not part of the device specification.
Unlinked/default values do not prove valid I/O. The caller evaluates bus/channel validity before use.
Use one owner task per instance and externally synchronize other access; multi-field snapshots are not atomic.
Copies store data without creating hardware links. Keep borrowed field references valid while consumers are bound.
This passive record performs no validation, synchronization, configuration or protocol advancement.
WcState=TRUE means process-data exchange is invalid. State is acyclic EtherCAT/link information,
not proof of current measurement validity. Link diagnostics to the matching slave InfoData entries.
The selected PDO representation is documented by the base terminal model.
InputToggle signals an input update by changing state; TRUE alone does not mean fresh data.
AdsAddr is acyclic mailbox addressing information, not a measurement-validity indicator.
</description>
*)
TYPE EL3403_EX EXTENDS EL3403 :
STRUCT
	WcState AT %I* : BOOL;
	InputToggle AT %I* : BOOL;
	State AT %I* : UINT;
	AdsAddr AT %I* : Global.AMSADDR;
END_STRUCT
END_TYPE

// ---- PowerMeasurement/EL3413/EL3413.TcDUT
(*
SPDX-FileCopyrightText: © 2026 Oleksandr Tiutyk <trofimich@gmail.com>
SPDX-License-Identifier: MIT
License: https://opensource.org/license/mit
*)

(*!
<summary>
Beckhoff EL3413: 3-phase power measurement terminal up to 690 V AC.
</summary>
<description>
Represents phase TxPDOs 0x1A00..0x1A02, auxiliary TxPDO 0x1A03,
phase selector RxPDOs 0x1600..0x1602 and auxiliary selector RxPDO 0x1603.
Phase and auxiliary Status fields are required; bit 14 invalidates the corresponding measurement.
Bus WcState and State do not replace measurement status. Interpret values using acknowledged input selectors.
Units and additional index selections follow firmware and configured transformer ratios.
Link fields individually. Use one owner task and synchronize other access; snapshots are not atomic.
When used for I/O, link located fields or their containing buffers to the matching selected PDOs.
The record is not a packed wire buffer; compiler padding is not part of the device specification.
Unlinked/default values do not prove valid I/O. The caller evaluates bus/channel validity before use.
Use one owner task per instance and externally synchronize other access; multi-field snapshots are not atomic.
Copies store data without creating hardware links. Keep borrowed field references valid while consumers are bound.
This passive record performs no validation, synchronization, configuration or protocol advancement.
</description>
*)
TYPE EL3413 :
STRUCT
	L1 : POWER_MEASUREMENT_CHANNEL;
	L2 : POWER_MEASUREMENT_CHANNEL;
	L3 : POWER_MEASUREMENT_CHANNEL;
	Auxiliary : POWER_MEASUREMENT_AUXILIARY_CHANNEL;
END_STRUCT
END_TYPE

// ---- PowerMeasurement/EL3413/EL3413_EX.TcDUT
(*
SPDX-FileCopyrightText: © 2026 Oleksandr Tiutyk <trofimich@gmail.com>
SPDX-License-Identifier: MIT
License: https://opensource.org/license/mit
*)

(*!
<summary>
Beckhoff EL3413_EX: Extended 3-phase power measurement terminal up to 690 V AC with diagnostics.
</summary>
<description>
Extends EL3413 with EtherCAT Working Counter, slave state, and CoE mailbox ADS address diagnostics.
When used for I/O, link located fields or their containing buffers to the matching selected PDOs.
The record is not a packed wire buffer; compiler padding is not part of the device specification.
Unlinked/default values do not prove valid I/O. The caller evaluates bus/channel validity before use.
Use one owner task per instance and externally synchronize other access; multi-field snapshots are not atomic.
Copies store data without creating hardware links. Keep borrowed field references valid while consumers are bound.
This passive record performs no validation, synchronization, configuration or protocol advancement.
WcState=TRUE means process-data exchange is invalid. State is acyclic EtherCAT/link information,
not proof of current measurement validity. Link diagnostics to the matching slave InfoData entries.
The selected PDO representation is documented by the base terminal model.
InputToggle signals an input update by changing state; TRUE alone does not mean fresh data.
AdsAddr is acyclic mailbox addressing information, not a measurement-validity indicator.
</description>
*)
TYPE EL3413_EX EXTENDS EL3413 :
STRUCT
	WcState AT %I* : BOOL;
	InputToggle AT %I* : BOOL;
	State AT %I* : UINT;
	AdsAddr AT %I* : Global.AMSADDR;
END_STRUCT
END_TYPE

// ---- PowerMeasurement/EL3433/EL3433.TcDUT
(*
SPDX-FileCopyrightText: © 2026 Oleksandr Tiutyk <trofimich@gmail.com>
SPDX-License-Identifier: MIT
License: https://opensource.org/license/mit
*)

(*!
<summary>
Beckhoff EL3433: 3-phase power measurement terminal with internal 10 A current measurement.
</summary>
<description>
Represents phase TxPDOs 0x1A00..0x1A02, auxiliary TxPDO 0x1A03,
phase selector RxPDOs 0x1600..0x1602 and auxiliary selector RxPDO 0x1603.
Phase and auxiliary Status fields are required; bit 14 invalidates the corresponding measurement.
Bus WcState and State do not replace measurement status. Interpret values using acknowledged input selectors.
Units and additional index selections follow firmware and configured transformer ratios.
Link fields individually. Use one owner task and synchronize other access; snapshots are not atomic.
When used for I/O, link located fields or their containing buffers to the matching selected PDOs.
The record is not a packed wire buffer; compiler padding is not part of the device specification.
Unlinked/default values do not prove valid I/O. The caller evaluates bus/channel validity before use.
Use one owner task per instance and externally synchronize other access; multi-field snapshots are not atomic.
Copies store data without creating hardware links. Keep borrowed field references valid while consumers are bound.
This passive record performs no validation, synchronization, configuration or protocol advancement.
</description>
*)
TYPE EL3433 :
STRUCT
	L1 : POWER_MEASUREMENT_CHANNEL;
	L2 : POWER_MEASUREMENT_CHANNEL;
	L3 : POWER_MEASUREMENT_CHANNEL;
	Auxiliary : POWER_MEASUREMENT_AUXILIARY_CHANNEL;
END_STRUCT
END_TYPE

// ---- PowerMeasurement/EL3433/EL3433_EX.TcDUT
(*
SPDX-FileCopyrightText: © 2026 Oleksandr Tiutyk <trofimich@gmail.com>
SPDX-License-Identifier: MIT
License: https://opensource.org/license/mit
*)

(*!
<summary>
Beckhoff EL3433_EX: Extended 3-phase power measurement terminal with internal 10 A current measurement with
diagnostics.
</summary>
<description>
Extends EL3433 with EtherCAT Working Counter, slave state, and CoE mailbox ADS address diagnostics.
When used for I/O, link located fields or their containing buffers to the matching selected PDOs.
The record is not a packed wire buffer; compiler padding is not part of the device specification.
Unlinked/default values do not prove valid I/O. The caller evaluates bus/channel validity before use.
Use one owner task per instance and externally synchronize other access; multi-field snapshots are not atomic.
Copies store data without creating hardware links. Keep borrowed field references valid while consumers are bound.
This passive record performs no validation, synchronization, configuration or protocol advancement.
WcState=TRUE means process-data exchange is invalid. State is acyclic EtherCAT/link information,
not proof of current measurement validity. Link diagnostics to the matching slave InfoData entries.
The selected PDO representation is documented by the base terminal model.
InputToggle signals an input update by changing state; TRUE alone does not mean fresh data.
AdsAddr is acyclic mailbox addressing information, not a measurement-validity indicator.
</description>
*)
TYPE EL3433_EX EXTENDS EL3433 :
STRUCT
	WcState AT %I* : BOOL;
	InputToggle AT %I* : BOOL;
	State AT %I* : UINT;
	AdsAddr AT %I* : Global.AMSADDR;
END_STRUCT
END_TYPE

// ---- DigitalIO/Inputs/EP1008_0001/EP1008_0001.TcDUT
(*
SPDX-FileCopyrightText: © 2026 Oleksandr Tiutyk <trofimich@gmail.com>
SPDX-License-Identifier: MIT
License: https://opensource.org/license/mit
*)

(*!
<summary>
Beckhoff EP1008_0001: 8-channel digital input EtherCAT Box (24 V DC, 3 ms filter, M8).
</summary>
<description>
Process image mapping structure for the EP1008_0001 EtherCAT Box IP67 module with 8 discrete inputs.
When used for I/O, link located fields or their containing buffers to the matching selected PDOs.
The record is not a packed wire buffer; compiler padding is not part of the device specification.
Unlinked/default values do not prove valid I/O. The caller evaluates bus/channel validity before use.
Use one owner task per instance and externally synchronize other access; multi-field snapshots are not atomic.
Copies store data without creating hardware links. Keep borrowed field references valid while consumers are bound.
This passive record performs no validation, synchronization, configuration or protocol advancement.
</description>
*)
TYPE EP1008_0001 :
STRUCT
	Ch1 AT %I* : BOOL;
	Ch2 AT %I* : BOOL;
	Ch3 AT %I* : BOOL;
	Ch4 AT %I* : BOOL;
	Ch5 AT %I* : BOOL;
	Ch6 AT %I* : BOOL;
	Ch7 AT %I* : BOOL;
	Ch8 AT %I* : BOOL;
END_STRUCT
END_TYPE

// ---- DigitalIO/Inputs/EP1008_0001/EP1008_0001_EX.TcDUT
(*
SPDX-FileCopyrightText: © 2026 Oleksandr Tiutyk <trofimich@gmail.com>
SPDX-License-Identifier: MIT
License: https://opensource.org/license/mit
*)

(*!
<summary>
Beckhoff EP1008_0001_EX: Extended 8-channel digital input EtherCAT Box (24 V DC, 3 ms filter, M8) with
diagnostics.
</summary>
<description>
Extends EP1008_0001 with EtherCAT Working Counter and slave state diagnostics.
This slave has no CoE mailbox; no ADS mailbox address endpoint is provided.
When used for I/O, link located fields or their containing buffers to the matching selected PDOs.
The record is not a packed wire buffer; compiler padding is not part of the device specification.
Unlinked/default values do not prove valid I/O. The caller evaluates bus/channel validity before use.
Use one owner task per instance and externally synchronize other access; multi-field snapshots are not atomic.
Copies store data without creating hardware links. Keep borrowed field references valid while consumers are bound.
This passive record performs no validation, synchronization, configuration or protocol advancement.
WcState=TRUE means process-data exchange is invalid. State is acyclic EtherCAT/link information,
not proof of current measurement validity. Link diagnostics to the matching slave InfoData entries.
The selected PDO representation is documented by the base terminal model.
InputToggle signals an input update by changing state; TRUE alone does not mean fresh data.
</description>
*)
TYPE EP1008_0001_EX EXTENDS EP1008_0001 :
STRUCT
	WcState AT %I* : BOOL;
	InputToggle AT %I* : BOOL;
	State AT %I* : UINT;
END_STRUCT
END_TYPE

// ---- DigitalIO/Inputs/EP1008_0002/EP1008_0002.TcDUT
(*
SPDX-FileCopyrightText: © 2026 Oleksandr Tiutyk <trofimich@gmail.com>
SPDX-License-Identifier: MIT
License: https://opensource.org/license/mit
*)

(*!
<summary>
Beckhoff EP1008_0002: 8-channel digital input EtherCAT Box (24 V DC, 3 ms filter, M12).
</summary>
<description>
Process image mapping structure for the EP1008_0002 EtherCAT Box IP67 module with 8 discrete inputs.
When used for I/O, link located fields or their containing buffers to the matching selected PDOs.
The record is not a packed wire buffer; compiler padding is not part of the device specification.
Unlinked/default values do not prove valid I/O. The caller evaluates bus/channel validity before use.
Use one owner task per instance and externally synchronize other access; multi-field snapshots are not atomic.
Copies store data without creating hardware links. Keep borrowed field references valid while consumers are bound.
This passive record performs no validation, synchronization, configuration or protocol advancement.
</description>
*)
TYPE EP1008_0002 :
STRUCT
	Ch1 AT %I* : BOOL;
	Ch2 AT %I* : BOOL;
	Ch3 AT %I* : BOOL;
	Ch4 AT %I* : BOOL;
	Ch5 AT %I* : BOOL;
	Ch6 AT %I* : BOOL;
	Ch7 AT %I* : BOOL;
	Ch8 AT %I* : BOOL;
END_STRUCT
END_TYPE

// ---- DigitalIO/Inputs/EP1008_0002/EP1008_0002_EX.TcDUT
(*
SPDX-FileCopyrightText: © 2026 Oleksandr Tiutyk <trofimich@gmail.com>
SPDX-License-Identifier: MIT
License: https://opensource.org/license/mit
*)

(*!
<summary>
Beckhoff EP1008_0002_EX: Extended 8-channel digital input EtherCAT Box (24 V DC, 3 ms filter, M12) with
diagnostics.
</summary>
<description>
Extends EP1008_0002 with EtherCAT Working Counter and slave state diagnostics.
This slave has no CoE mailbox; no ADS mailbox address endpoint is provided.
When used for I/O, link located fields or their containing buffers to the matching selected PDOs.
The record is not a packed wire buffer; compiler padding is not part of the device specification.
Unlinked/default values do not prove valid I/O. The caller evaluates bus/channel validity before use.
Use one owner task per instance and externally synchronize other access; multi-field snapshots are not atomic.
Copies store data without creating hardware links. Keep borrowed field references valid while consumers are bound.
This passive record performs no validation, synchronization, configuration or protocol advancement.
WcState=TRUE means process-data exchange is invalid. State is acyclic EtherCAT/link information,
not proof of current measurement validity. Link diagnostics to the matching slave InfoData entries.
The selected PDO representation is documented by the base terminal model.
InputToggle signals an input update by changing state; TRUE alone does not mean fresh data.
</description>
*)
TYPE EP1008_0002_EX EXTENDS EP1008_0002 :
STRUCT
	WcState AT %I* : BOOL;
	InputToggle AT %I* : BOOL;
	State AT %I* : UINT;
END_STRUCT
END_TYPE

// ---- DigitalIO/Inputs/EP1018_0001/EP1018_0001.TcDUT
(*
SPDX-FileCopyrightText: © 2026 Oleksandr Tiutyk <trofimich@gmail.com>
SPDX-License-Identifier: MIT
License: https://opensource.org/license/mit
*)

(*!
<summary>
Beckhoff EP1018_0001: 8-channel digital input EtherCAT Box (24 V DC, 10 µs filter, M8).
</summary>
<description>
Process image mapping structure for the EP1018_0001 EtherCAT Box IP67 module with 8 discrete inputs.
When used for I/O, link located fields or their containing buffers to the matching selected PDOs.
The record is not a packed wire buffer; compiler padding is not part of the device specification.
Unlinked/default values do not prove valid I/O. The caller evaluates bus/channel validity before use.
Use one owner task per instance and externally synchronize other access; multi-field snapshots are not atomic.
Copies store data without creating hardware links. Keep borrowed field references valid while consumers are bound.
This passive record performs no validation, synchronization, configuration or protocol advancement.
</description>
*)
TYPE EP1018_0001 :
STRUCT
	Ch1 AT %I* : BOOL;
	Ch2 AT %I* : BOOL;
	Ch3 AT %I* : BOOL;
	Ch4 AT %I* : BOOL;
	Ch5 AT %I* : BOOL;
	Ch6 AT %I* : BOOL;
	Ch7 AT %I* : BOOL;
	Ch8 AT %I* : BOOL;
END_STRUCT
END_TYPE

// ---- DigitalIO/Inputs/EP1018_0001/EP1018_0001_EX.TcDUT
(*
SPDX-FileCopyrightText: © 2026 Oleksandr Tiutyk <trofimich@gmail.com>
SPDX-License-Identifier: MIT
License: https://opensource.org/license/mit
*)

(*!
<summary>
Beckhoff EP1018_0001_EX: Extended 8-channel digital input EtherCAT Box (24 V DC, 10 µs filter, M8) with
diagnostics.
</summary>
<description>
Extends EP1018_0001 with EtherCAT Working Counter and slave state diagnostics.
This slave has no CoE mailbox; no ADS mailbox address endpoint is provided.
When used for I/O, link located fields or their containing buffers to the matching selected PDOs.
The record is not a packed wire buffer; compiler padding is not part of the device specification.
Unlinked/default values do not prove valid I/O. The caller evaluates bus/channel validity before use.
Use one owner task per instance and externally synchronize other access; multi-field snapshots are not atomic.
Copies store data without creating hardware links. Keep borrowed field references valid while consumers are bound.
This passive record performs no validation, synchronization, configuration or protocol advancement.
WcState=TRUE means process-data exchange is invalid. State is acyclic EtherCAT/link information,
not proof of current measurement validity. Link diagnostics to the matching slave InfoData entries.
The selected PDO representation is documented by the base terminal model.
InputToggle signals an input update by changing state; TRUE alone does not mean fresh data.
</description>
*)
TYPE EP1018_0001_EX EXTENDS EP1018_0001 :
STRUCT
	WcState AT %I* : BOOL;
	InputToggle AT %I* : BOOL;
	State AT %I* : UINT;
END_STRUCT
END_TYPE

// ---- DigitalIO/Inputs/EP1809_0021/EP1809_0021.TcDUT
(*
SPDX-FileCopyrightText: © 2026 Oleksandr Tiutyk <trofimich@gmail.com>
SPDX-License-Identifier: MIT
License: https://opensource.org/license/mit
*)

(*!
<summary>
Beckhoff EP1809_0021: 16-channel digital input EtherCAT Box (24 V DC, 3 ms filter, M8).
</summary>
<description>
Process image mapping structure for the EP1809_0021 EtherCAT Box IP67 module with 16 discrete inputs.
When used for I/O, link located fields or their containing buffers to the matching selected PDOs.
The record is not a packed wire buffer; compiler padding is not part of the device specification.
Unlinked/default values do not prove valid I/O. The caller evaluates bus/channel validity before use.
Use one owner task per instance and externally synchronize other access; multi-field snapshots are not atomic.
Copies store data without creating hardware links. Keep borrowed field references valid while consumers are bound.
This passive record performs no validation, synchronization, configuration or protocol advancement.
</description>
*)
TYPE EP1809_0021 :
STRUCT
	Ch01 AT %I* : BOOL;
	Ch02 AT %I* : BOOL;
	Ch03 AT %I* : BOOL;
	Ch04 AT %I* : BOOL;
	Ch05 AT %I* : BOOL;
	Ch06 AT %I* : BOOL;
	Ch07 AT %I* : BOOL;
	Ch08 AT %I* : BOOL;
	Ch09 AT %I* : BOOL;
	Ch10 AT %I* : BOOL;
	Ch11 AT %I* : BOOL;
	Ch12 AT %I* : BOOL;
	Ch13 AT %I* : BOOL;
	Ch14 AT %I* : BOOL;
	Ch15 AT %I* : BOOL;
	Ch16 AT %I* : BOOL;
END_STRUCT
END_TYPE

// ---- DigitalIO/Inputs/EP1809_0021/EP1809_0021_EX.TcDUT
(*
SPDX-FileCopyrightText: © 2026 Oleksandr Tiutyk <trofimich@gmail.com>
SPDX-License-Identifier: MIT
License: https://opensource.org/license/mit
*)

(*!
<summary>
Beckhoff EP1809_0021_EX: Extended 16-channel digital input EtherCAT Box (24 V DC, 3 ms filter, M8) with
diagnostics.
</summary>
<description>
Extends EP1809_0021 with EtherCAT Working Counter and slave state diagnostics.
This slave has no CoE mailbox; no ADS mailbox address endpoint is provided.
When used for I/O, link located fields or their containing buffers to the matching selected PDOs.
The record is not a packed wire buffer; compiler padding is not part of the device specification.
Unlinked/default values do not prove valid I/O. The caller evaluates bus/channel validity before use.
Use one owner task per instance and externally synchronize other access; multi-field snapshots are not atomic.
Copies store data without creating hardware links. Keep borrowed field references valid while consumers are bound.
This passive record performs no validation, synchronization, configuration or protocol advancement.
WcState=TRUE means process-data exchange is invalid. State is acyclic EtherCAT/link information,
not proof of current measurement validity. Link diagnostics to the matching slave InfoData entries.
The selected PDO representation is documented by the base terminal model.
InputToggle signals an input update by changing state; TRUE alone does not mean fresh data.
</description>
*)
TYPE EP1809_0021_EX EXTENDS EP1809_0021 :
STRUCT
	WcState AT %I* : BOOL;
	InputToggle AT %I* : BOOL;
	State AT %I* : UINT;
END_STRUCT
END_TYPE

// ---- DigitalIO/Outputs/EP2008_0001/EP2008_0001.TcDUT
(*
SPDX-FileCopyrightText: © 2026 Oleksandr Tiutyk <trofimich@gmail.com>
SPDX-License-Identifier: MIT
License: https://opensource.org/license/mit
*)

(*!
<summary>
Beckhoff EP2008_0001: 8-channel digital output EtherCAT Box (24 V DC, 0.5 A, M8).
</summary>
<description>
Process image mapping structure for the EP2008_0001 EtherCAT Box IP67 module with 8 discrete outputs.
When used for I/O, link located fields or their containing buffers to the matching selected PDOs.
The record is not a packed wire buffer; compiler padding is not part of the device specification.
Unlinked/default values do not prove valid I/O. The caller evaluates bus/channel validity before use.
Use one owner task per instance and externally synchronize other access; multi-field snapshots are not atomic.
Copies store data without creating hardware links. Keep borrowed field references valid while consumers are bound.
This passive record performs no validation, synchronization, configuration or protocol advancement.
</description>
*)
TYPE EP2008_0001 :
STRUCT
	Ch1 AT %Q* : BOOL;
	Ch2 AT %Q* : BOOL;
	Ch3 AT %Q* : BOOL;
	Ch4 AT %Q* : BOOL;
	Ch5 AT %Q* : BOOL;
	Ch6 AT %Q* : BOOL;
	Ch7 AT %Q* : BOOL;
	Ch8 AT %Q* : BOOL;
END_STRUCT
END_TYPE

// ---- DigitalIO/Outputs/EP2008_0001/EP2008_0001_EX.TcDUT
(*
SPDX-FileCopyrightText: © 2026 Oleksandr Tiutyk <trofimich@gmail.com>
SPDX-License-Identifier: MIT
License: https://opensource.org/license/mit
*)

(*!
<summary>
Beckhoff EP2008_0001_EX: Extended 8-channel digital output EtherCAT Box (24 V DC, 0.5 A, M8) with diagnostics.
</summary>
<description>
Extends EP2008_0001 with EtherCAT Working Counter and slave state diagnostics.
This slave has no CoE mailbox; no ADS mailbox address endpoint is provided.
When used for I/O, link located fields or their containing buffers to the matching selected PDOs.
The record is not a packed wire buffer; compiler padding is not part of the device specification.
Unlinked/default values do not prove valid I/O. The caller evaluates bus/channel validity before use.
Use one owner task per instance and externally synchronize other access; multi-field snapshots are not atomic.
Copies store data without creating hardware links. Keep borrowed field references valid while consumers are bound.
This passive record performs no validation, synchronization, configuration or protocol advancement.
WcState=TRUE means process-data exchange is invalid. State is acyclic EtherCAT/link information,
not proof of current measurement validity. Link diagnostics to the matching slave InfoData entries.
The selected PDO representation is documented by the base terminal model.
</description>
*)
TYPE EP2008_0001_EX EXTENDS EP2008_0001 :
STRUCT
	WcState AT %I* : BOOL;
	State AT %I* : UINT;
END_STRUCT
END_TYPE

// ---- DigitalIO/Outputs/EP2008_0002/EP2008_0002.TcDUT
(*
SPDX-FileCopyrightText: © 2026 Oleksandr Tiutyk <trofimich@gmail.com>
SPDX-License-Identifier: MIT
License: https://opensource.org/license/mit
*)

(*!
<summary>
Beckhoff EP2008_0002: 8-channel digital output EtherCAT Box (24 V DC, 0.5 A, M12).
</summary>
<description>
Process image mapping structure for the EP2008_0002 EtherCAT Box IP67 module with 8 discrete outputs.
When used for I/O, link located fields or their containing buffers to the matching selected PDOs.
The record is not a packed wire buffer; compiler padding is not part of the device specification.
Unlinked/default values do not prove valid I/O. The caller evaluates bus/channel validity before use.
Use one owner task per instance and externally synchronize other access; multi-field snapshots are not atomic.
Copies store data without creating hardware links. Keep borrowed field references valid while consumers are bound.
This passive record performs no validation, synchronization, configuration or protocol advancement.
</description>
*)
TYPE EP2008_0002 :
STRUCT
	Ch1 AT %Q* : BOOL;
	Ch2 AT %Q* : BOOL;
	Ch3 AT %Q* : BOOL;
	Ch4 AT %Q* : BOOL;
	Ch5 AT %Q* : BOOL;
	Ch6 AT %Q* : BOOL;
	Ch7 AT %Q* : BOOL;
	Ch8 AT %Q* : BOOL;
END_STRUCT
END_TYPE

// ---- DigitalIO/Outputs/EP2008_0002/EP2008_0002_EX.TcDUT
(*
SPDX-FileCopyrightText: © 2026 Oleksandr Tiutyk <trofimich@gmail.com>
SPDX-License-Identifier: MIT
License: https://opensource.org/license/mit
*)

(*!
<summary>
Beckhoff EP2008_0002_EX: Extended 8-channel digital output EtherCAT Box (24 V DC, 0.5 A, M12) with
diagnostics.
</summary>
<description>
Extends EP2008_0002 with EtherCAT Working Counter and slave state diagnostics.
This slave has no CoE mailbox; no ADS mailbox address endpoint is provided.
When used for I/O, link located fields or their containing buffers to the matching selected PDOs.
The record is not a packed wire buffer; compiler padding is not part of the device specification.
Unlinked/default values do not prove valid I/O. The caller evaluates bus/channel validity before use.
Use one owner task per instance and externally synchronize other access; multi-field snapshots are not atomic.
Copies store data without creating hardware links. Keep borrowed field references valid while consumers are bound.
This passive record performs no validation, synchronization, configuration or protocol advancement.
WcState=TRUE means process-data exchange is invalid. State is acyclic EtherCAT/link information,
not proof of current measurement validity. Link diagnostics to the matching slave InfoData entries.
The selected PDO representation is documented by the base terminal model.
</description>
*)
TYPE EP2008_0002_EX EXTENDS EP2008_0002 :
STRUCT
	WcState AT %I* : BOOL;
	State AT %I* : UINT;
END_STRUCT
END_TYPE

// ---- DigitalIO/Outputs/EP2809_0021/EP2809_0021.TcDUT
(*
SPDX-FileCopyrightText: © 2026 Oleksandr Tiutyk <trofimich@gmail.com>
SPDX-License-Identifier: MIT
License: https://opensource.org/license/mit
*)

(*!
<summary>
Beckhoff EP2809_0021: 16-channel digital output EtherCAT Box (24 V DC, 0.5 A, M8).
</summary>
<description>
Process image mapping structure for the EP2809_0021 EtherCAT Box IP67 module with 16 discrete outputs.
When used for I/O, link located fields or their containing buffers to the matching selected PDOs.
The record is not a packed wire buffer; compiler padding is not part of the device specification.
Unlinked/default values do not prove valid I/O. The caller evaluates bus/channel validity before use.
Use one owner task per instance and externally synchronize other access; multi-field snapshots are not atomic.
Copies store data without creating hardware links. Keep borrowed field references valid while consumers are bound.
This passive record performs no validation, synchronization, configuration or protocol advancement.
</description>
*)
TYPE EP2809_0021 :
STRUCT
	Ch01 AT %Q* : BOOL;
	Ch02 AT %Q* : BOOL;
	Ch03 AT %Q* : BOOL;
	Ch04 AT %Q* : BOOL;
	Ch05 AT %Q* : BOOL;
	Ch06 AT %Q* : BOOL;
	Ch07 AT %Q* : BOOL;
	Ch08 AT %Q* : BOOL;
	Ch09 AT %Q* : BOOL;
	Ch10 AT %Q* : BOOL;
	Ch11 AT %Q* : BOOL;
	Ch12 AT %Q* : BOOL;
	Ch13 AT %Q* : BOOL;
	Ch14 AT %Q* : BOOL;
	Ch15 AT %Q* : BOOL;
	Ch16 AT %Q* : BOOL;
END_STRUCT
END_TYPE

// ---- DigitalIO/Outputs/EP2809_0021/EP2809_0021_EX.TcDUT
(*
SPDX-FileCopyrightText: © 2026 Oleksandr Tiutyk <trofimich@gmail.com>
SPDX-License-Identifier: MIT
License: https://opensource.org/license/mit
*)

(*!
<summary>
Beckhoff EP2809_0021_EX: Extended 16-channel digital output EtherCAT Box (24 V DC, 0.5 A, M8) with
diagnostics.
</summary>
<description>
Extends EP2809_0021 with EtherCAT Working Counter and slave state diagnostics.
This slave has no CoE mailbox; no ADS mailbox address endpoint is provided.
When used for I/O, link located fields or their containing buffers to the matching selected PDOs.
The record is not a packed wire buffer; compiler padding is not part of the device specification.
Unlinked/default values do not prove valid I/O. The caller evaluates bus/channel validity before use.
Use one owner task per instance and externally synchronize other access; multi-field snapshots are not atomic.
Copies store data without creating hardware links. Keep borrowed field references valid while consumers are bound.
This passive record performs no validation, synchronization, configuration or protocol advancement.
WcState=TRUE means process-data exchange is invalid. State is acyclic EtherCAT/link information,
not proof of current measurement validity. Link diagnostics to the matching slave InfoData entries.
The selected PDO representation is documented by the base terminal model.
</description>
*)
TYPE EP2809_0021_EX EXTENDS EP2809_0021 :
STRUCT
	WcState AT %I* : BOOL;
	State AT %I* : UINT;
END_STRUCT
END_TYPE

// ---- DigitalIO/Outputs/EP2624_0002/EP2624_0002.TcDUT
(*
SPDX-FileCopyrightText: © 2026 Oleksandr Tiutyk <trofimich@gmail.com>
SPDX-License-Identifier: MIT
License: https://opensource.org/license/mit
*)

(*!
<summary>
Beckhoff EP2624_0002: 4-channel relay output EtherCAT Box (25 V AC / 30 V DC, make/NO contact, M12).
</summary>
<description>
Process image mapping structure for the EP2624_0002 EtherCAT Box IP67 module with 4 discrete outputs.
The relay ratings are 0.5 A AC at 25 V AC and 2 A DC at 30 V DC; this is not a 230 V AC relay module.
When used for I/O, link located fields or their containing buffers to the matching selected PDOs.
The record is not a packed wire buffer; compiler padding is not part of the device specification.
Unlinked/default values do not prove valid I/O. The caller evaluates bus/channel validity before use.
Use one owner task per instance and externally synchronize other access; multi-field snapshots are not atomic.
Copies store data without creating hardware links. Keep borrowed field references valid while consumers are bound.
This passive record performs no validation, synchronization, configuration or protocol advancement.
</description>
*)
TYPE EP2624_0002 :
STRUCT
	Ch1 AT %Q* : BOOL;
	Ch2 AT %Q* : BOOL;
	Ch3 AT %Q* : BOOL;
	Ch4 AT %Q* : BOOL;
END_STRUCT
END_TYPE

// ---- DigitalIO/Outputs/EP2624_0002/EP2624_0002_EX.TcDUT
(*
SPDX-FileCopyrightText: © 2026 Oleksandr Tiutyk <trofimich@gmail.com>
SPDX-License-Identifier: MIT
License: https://opensource.org/license/mit
*)

(*!
<summary>
Beckhoff EP2624_0002_EX: Extended 4-channel relay output EtherCAT Box (25 V AC / 30 V DC, make/NO contact,
M12) with diagnostics.
</summary>
<description>
Extends EP2624_0002 with EtherCAT Working Counter and slave state diagnostics.
This slave has no CoE mailbox; no ADS mailbox address endpoint is provided.
Relay ratings are 0.5 A AC at 25 V AC and 2 A DC at 30 V DC.
When used for I/O, link located fields or their containing buffers to the matching selected PDOs.
The record is not a packed wire buffer; compiler padding is not part of the device specification.
Unlinked/default values do not prove valid I/O. The caller evaluates bus/channel validity before use.
Use one owner task per instance and externally synchronize other access; multi-field snapshots are not atomic.
Copies store data without creating hardware links. Keep borrowed field references valid while consumers are bound.
This passive record performs no validation, synchronization, configuration or protocol advancement.
WcState=TRUE means process-data exchange is invalid. State is acyclic EtherCAT/link information,
not proof of current measurement validity. Link diagnostics to the matching slave InfoData entries.
The selected PDO representation is documented by the base terminal model.
</description>
*)
TYPE EP2624_0002_EX EXTENDS EP2624_0002 :
STRUCT
	WcState AT %I* : BOOL;
	State AT %I* : UINT;
END_STRUCT
END_TYPE

// ---- AnalogIO/Inputs/EP3174_0002/EP3174_0002.TcDUT
(*
SPDX-FileCopyrightText: © 2026 Oleksandr Tiutyk <trofimich@gmail.com>
SPDX-License-Identifier: MIT
License: https://opensource.org/license/mit
*)

(*!
<summary>
Beckhoff EP3174-0002: 4-channel configurable analog input EtherCAT Box (-10..+10 V, 0/4..20 mA, 16-bit, M12).
</summary>
<description>
Process image mapping structure for the EP3174-0002 EtherCAT Box IP67 module with 4 multi-range analog inputs.
When used for I/O, link located fields or their containing buffers to the matching selected PDOs.
The record is not a packed wire buffer; compiler padding is not part of the device specification.
Unlinked/default values do not prove valid I/O. The caller evaluates bus/channel validity before use.
Use one owner task per instance and externally synchronize other access; multi-field snapshots are not atomic.
Copies store data without creating hardware links. Keep borrowed field references valid while consumers are bound.
This passive record performs no validation, synchronization, configuration or protocol advancement.
Select standard status-plus-value PDOs matching the declared Value type; compact value-only PDOs
are outside this model. Configure electrical range and scaling separately on the device.
</description>
*)
TYPE EP3174_0002 :
STRUCT
	Ch1 : ANALOG_INPUT_INT_CHANNEL;
	Ch2 : ANALOG_INPUT_INT_CHANNEL;
	Ch3 : ANALOG_INPUT_INT_CHANNEL;
	Ch4 : ANALOG_INPUT_INT_CHANNEL;
END_STRUCT
END_TYPE

// ---- AnalogIO/Inputs/EP3174_0002/EP3174_0002_EX.TcDUT
(*
SPDX-FileCopyrightText: © 2026 Oleksandr Tiutyk <trofimich@gmail.com>
SPDX-License-Identifier: MIT
License: https://opensource.org/license/mit
*)

(*!
<summary>
Beckhoff EP3174_0002_EX: Extended 4-channel configurable analog input EtherCAT Box with diagnostics.
</summary>
<description>
Extends EP3174_0002 with EtherCAT Working Counter, slave state, and CoE mailbox ADS address diagnostics.
When used for I/O, link located fields or their containing buffers to the matching selected PDOs.
The record is not a packed wire buffer; compiler padding is not part of the device specification.
Unlinked/default values do not prove valid I/O. The caller evaluates bus/channel validity before use.
Use one owner task per instance and externally synchronize other access; multi-field snapshots are not atomic.
Copies store data without creating hardware links. Keep borrowed field references valid while consumers are bound.
This passive record performs no validation, synchronization, configuration or protocol advancement.
WcState=TRUE means process-data exchange is invalid. State is acyclic EtherCAT/link information,
not proof of current measurement validity. Link diagnostics to the matching slave InfoData entries.
The selected PDO representation is documented by the base terminal model.
InputToggle signals an input update by changing state; TRUE alone does not mean fresh data.
AdsAddr is acyclic mailbox addressing information, not a measurement-validity indicator.
Select standard status-plus-value PDOs matching the declared Value type; compact value-only PDOs
are outside this model. Configure electrical range and scaling separately on the device.
</description>
*)
TYPE EP3174_0002_EX EXTENDS EP3174_0002 :
STRUCT
	WcState AT %I* : BOOL;
	InputToggle AT %I* : BOOL;
	State AT %I* : UINT;
	AdsAddr AT %I* : Global.AMSADDR;
END_STRUCT
END_TYPE

// ---- AnalogIO/Outputs/EP4174_0002/EP4174_0002.TcDUT
(*
SPDX-FileCopyrightText: © 2026 Oleksandr Tiutyk <trofimich@gmail.com>
SPDX-License-Identifier: MIT
License: https://opensource.org/license/mit
*)

(*!
<summary>
Beckhoff EP4174-0002: 4-channel configurable analog output EtherCAT Box (-10..+10 V, 0/4..20 mA, 16-bit, M12).
</summary>
<description>
Process image mapping structure for the EP4174-0002 EtherCAT Box IP67 module with 4 multi-range analog
outputs.
When used for I/O, link located fields or their containing buffers to the matching selected PDOs.
The record is not a packed wire buffer; compiler padding is not part of the device specification.
Unlinked/default values do not prove valid I/O. The caller evaluates bus/channel validity before use.
Use one owner task per instance and externally synchronize other access; multi-field snapshots are not atomic.
Copies store data without creating hardware links. Keep borrowed field references valid while consumers are bound.
This passive record performs no validation, synchronization, configuration or protocol advancement.
Channels hold raw INT16 output commands; configure electrical range and presentation before use.
</description>
*)
TYPE EP4174_0002 :
STRUCT
	Ch1 AT %Q* : INT;
	Ch2 AT %Q* : INT;
	Ch3 AT %Q* : INT;
	Ch4 AT %Q* : INT;
END_STRUCT
END_TYPE

// ---- AnalogIO/Outputs/EP4174_0002/EP4174_0002_EX.TcDUT
(*
SPDX-FileCopyrightText: © 2026 Oleksandr Tiutyk <trofimich@gmail.com>
SPDX-License-Identifier: MIT
License: https://opensource.org/license/mit
*)

(*!
<summary>
Beckhoff EP4174_0002_EX: Extended 4-channel configurable analog output EtherCAT Box with diagnostics.
</summary>
<description>
Extends EP4174_0002 with EtherCAT Working Counter, slave state, and CoE mailbox ADS address diagnostics.
When used for I/O, link located fields or their containing buffers to the matching selected PDOs.
The record is not a packed wire buffer; compiler padding is not part of the device specification.
Unlinked/default values do not prove valid I/O. The caller evaluates bus/channel validity before use.
Use one owner task per instance and externally synchronize other access; multi-field snapshots are not atomic.
Copies store data without creating hardware links. Keep borrowed field references valid while consumers are bound.
This passive record performs no validation, synchronization, configuration or protocol advancement.
WcState=TRUE means process-data exchange is invalid. State is acyclic EtherCAT/link information,
not proof of current measurement validity. Link diagnostics to the matching slave InfoData entries.
The selected PDO representation is documented by the base terminal model.
AdsAddr is acyclic mailbox addressing information, not a measurement-validity indicator.
Channels hold raw INT16 output commands; configure electrical range and presentation before use.
</description>
*)
TYPE EP4174_0002_EX EXTENDS EP4174_0002 :
STRUCT
	WcState AT %I* : BOOL;
	State AT %I* : UINT;
	AdsAddr AT %I* : Global.AMSADDR;
END_STRUCT
END_TYPE

// ---- Serial/EP6001_0002/EP6001_0002.TcDUT
(*
SPDX-FileCopyrightText: © 2026 Oleksandr Tiutyk <trofimich@gmail.com>
SPDX-License-Identifier: MIT
License: https://opensource.org/license/mit
*)

(*!
<summary>
Beckhoff EP6001-0002: 1-channel serial interface EtherCAT Box (selectable RS232/RS422/RS485, M12).
</summary>
<description>
Represents one 22-byte serial channel. Configure RS232/RS422/RS485 independently on the device.
Optional digital I/O is outside this model; link it separately if enabled.
When used for I/O, link located fields or their containing buffers to the matching selected PDOs.
The record is not a packed wire buffer; compiler padding is not part of the device specification.
Unlinked/default values do not prove valid I/O. The caller evaluates bus/channel validity before use.
Use one owner task per instance and externally synchronize other access; multi-field snapshots are not atomic.
Copies store data without creating hardware links. Keep borrowed field references valid while consumers are bound.
This passive record performs no validation, synchronization, configuration or protocol advancement.
Select the 22-byte serial payload with 16-bit status/control words; larger buffers and 9-bit modes
are outside this model. The owning service implements the transmit/receive toggle handshake.
</description>
*)
TYPE EP6001_0002 :
STRUCT
	Ch1 : EL6022_CHANNEL;
END_STRUCT
END_TYPE

// ---- Serial/EP6001_0002/EP6001_0002_EX.TcDUT
(*
SPDX-FileCopyrightText: © 2026 Oleksandr Tiutyk <trofimich@gmail.com>
SPDX-License-Identifier: MIT
License: https://opensource.org/license/mit
*)

(*!
<summary>
Beckhoff EP6001_0002_EX: Extended 1-channel serial interface EtherCAT Box with diagnostics.
</summary>
<description>
Extends EP6001_0002 with EtherCAT Working Counter, slave state, and CoE mailbox ADS address diagnostics.
When used for I/O, link located fields or their containing buffers to the matching selected PDOs.
The record is not a packed wire buffer; compiler padding is not part of the device specification.
Unlinked/default values do not prove valid I/O. The caller evaluates bus/channel validity before use.
Use one owner task per instance and externally synchronize other access; multi-field snapshots are not atomic.
Copies store data without creating hardware links. Keep borrowed field references valid while consumers are bound.
This passive record performs no validation, synchronization, configuration or protocol advancement.
WcState=TRUE means process-data exchange is invalid. State is acyclic EtherCAT/link information,
not proof of current measurement validity. Link diagnostics to the matching slave InfoData entries.
The selected PDO representation is documented by the base terminal model.
InputToggle signals an input update by changing state; TRUE alone does not mean fresh data.
AdsAddr is acyclic mailbox addressing information, not a measurement-validity indicator.
Select the 22-byte serial payload with 16-bit status/control words; larger buffers and 9-bit modes
are outside this model. The owning service implements the transmit/receive toggle handshake.
</description>
*)
TYPE EP6001_0002_EX EXTENDS EP6001_0002 :
STRUCT
	WcState AT %I* : BOOL;
	InputToggle AT %I* : BOOL;
	State AT %I* : UINT;
	AdsAddr AT %I* : Global.AMSADDR;
END_STRUCT
END_TYPE

// ---- Serial/EP6002_0002/EP6002_0002.TcDUT
(*
SPDX-FileCopyrightText: © 2026 Oleksandr Tiutyk <trofimich@gmail.com>
SPDX-License-Identifier: MIT
License: https://opensource.org/license/mit
*)

(*!
<summary>
Beckhoff EP6002-0002: 2-channel serial interface EtherCAT Box (selectable RS232/RS422/RS485, M12).
</summary>
<description>
Represents two 22-byte serial channels. Configure RS232/RS422/RS485 independently on the device.
Larger serial process images are outside this model.
When used for I/O, link located fields or their containing buffers to the matching selected PDOs.
The record is not a packed wire buffer; compiler padding is not part of the device specification.
Unlinked/default values do not prove valid I/O. The caller evaluates bus/channel validity before use.
Use one owner task per instance and externally synchronize other access; multi-field snapshots are not atomic.
Copies store data without creating hardware links. Keep borrowed field references valid while consumers are bound.
This passive record performs no validation, synchronization, configuration or protocol advancement.
Select the 22-byte serial payload with 16-bit status/control words; larger buffers and 9-bit modes
are outside this model. The owning service implements the transmit/receive toggle handshake.
</description>
*)
TYPE EP6002_0002 :
STRUCT
	Ch1 : EL6022_CHANNEL;
	Ch2 : EL6022_CHANNEL;
END_STRUCT
END_TYPE

// ---- Serial/EP6002_0002/EP6002_0002_EX.TcDUT
(*
SPDX-FileCopyrightText: © 2026 Oleksandr Tiutyk <trofimich@gmail.com>
SPDX-License-Identifier: MIT
License: https://opensource.org/license/mit
*)

(*!
<summary>
Beckhoff EP6002_0002_EX: Extended 2-channel serial interface EtherCAT Box with diagnostics.
</summary>
<description>
Extends EP6002_0002 with EtherCAT Working Counter, slave state, and CoE mailbox ADS address diagnostics.
When used for I/O, link located fields or their containing buffers to the matching selected PDOs.
The record is not a packed wire buffer; compiler padding is not part of the device specification.
Unlinked/default values do not prove valid I/O. The caller evaluates bus/channel validity before use.
Use one owner task per instance and externally synchronize other access; multi-field snapshots are not atomic.
Copies store data without creating hardware links. Keep borrowed field references valid while consumers are bound.
This passive record performs no validation, synchronization, configuration or protocol advancement.
WcState=TRUE means process-data exchange is invalid. State is acyclic EtherCAT/link information,
not proof of current measurement validity. Link diagnostics to the matching slave InfoData entries.
The selected PDO representation is documented by the base terminal model.
InputToggle signals an input update by changing state; TRUE alone does not mean fresh data.
AdsAddr is acyclic mailbox addressing information, not a measurement-validity indicator.
Select the 22-byte serial payload with 16-bit status/control words; larger buffers and 9-bit modes
are outside this model. The owning service implements the transmit/receive toggle handshake.
</description>
*)
TYPE EP6002_0002_EX EXTENDS EP6002_0002 :
STRUCT
	WcState AT %I* : BOOL;
	InputToggle AT %I* : BOOL;
	State AT %I* : UINT;
	AdsAddr AT %I* : Global.AMSADDR;
END_STRUCT
END_TYPE

// ---- Version/Global_Version.TcGVL
{attribute 'TcGenerated'}
{attribute 'no-analysis'}
{attribute 'linkalways'}
// This function has been automatically generated from the project information.
VAR_GLOBAL CONSTANT
	{attribute 'const_non_replaced'}
	stLibVersion_TwinCAT_Open_Framework_IO_Models : ST_LibVersion := (iMajor := 1, iMinor := 0, iBuild := 13, iRevision := 0, nFlags := 0, sVersion := '1.0.13.0');
END_VAR

// ---- Internal/CurrentNamespace.TcPOU
(*
SPDX-FileCopyrightText: © 2026 Oleksandr Tiutyk <trofimich@gmail.com>
SPDX-License-Identifier: MIT
License: https://opensource.org/license/mit
*)

(*!
<summary>
Internal service program providing access to the current library namespace.
</summary>
*)

{attribute 'no_explicit_call' := 'do not call this POU directly'}
PROGRAM INTERNAL CurrentNamespace
VAR
	{attribute 'hide'} 
	_NamespaceExtractor : NamespaceExtractor;
END_VAR

(*!
<summary>Borrows the compiler-initialized namespace buffer for the program lifetime.</summary>
<description>
Callers must not modify or retain the reference beyond the program lifetime. A reference property remains
technically writable without a setter; read-only use is a caller obligation. No allocation or initialization occurs.
</description>
*)
{attribute 'monitoring' := 'call'}
PROPERTY Name : REFERENCE TO STRING
GET
Name REF= _NamespaceExtractor.CurrentNamespace;
END_GET
END_PROPERTY

END_PROGRAM

// ---- Internal/NamespaceExtractor.TcPOU
(*
SPDX-FileCopyrightText: © 2026 Oleksandr Tiutyk <trofimich@gmail.com>
SPDX-License-Identifier: MIT
License: https://opensource.org/license/mit
*)

(*!
<summary>
Internal helper function block extracting library namespace via attribute init_namespace.
</summary>
*)

FUNCTION_BLOCK INTERNAL NamespaceExtractor
VAR_OUTPUT
	{attribute 'init_namespace'} 
	CurrentNamespace : STRING; 	
END_VAR

END_FUNCTION_BLOCK
